Universal Robots PolyScope program: weigh_touch3.urp

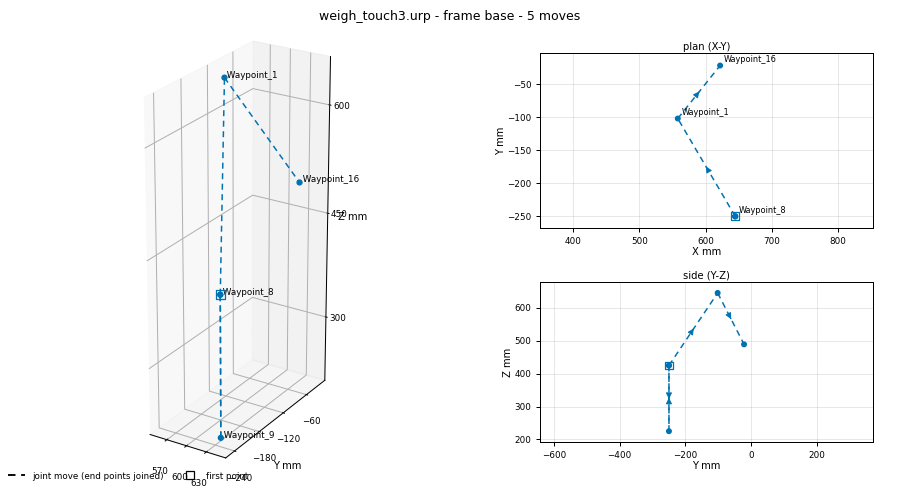
[picture p0: tool path of weigh_touch3.urp in frame base, 5 of 5 moves have a stored position in this frame; points joined in program order, loops and branches not executed]
Program weigh_touch3 (installation=default directory=/programs/Nicolas_Arteaga/quality createdIn=5.8.2.10297 lastSavedIn=5.12.4.1101661 robotSerialNumber=20225502378)
Calibrated DH parameters: a=[0.00022, -0.425328, -0.389701, 0.000059, 0.000065, 0]; d=[0.162608, 0.803456, 9.992211, -10.662202, 0.099702, 0.099559]; alpha=[1.570756, 0.001543, 0.004316, 1.570651, -1.570122, 0]; deltaTheta=[0, 0.002917, 0.116094, -0.119008, 0, -0.000001]
Robot Program (runOnlyOnce=true)
  MoveJ speed 60 deg/s, acceleration 80 deg/s^2 (useActiveTCP=true) feature=Base
    Waypoint Waypoint_8: TCP in base x=644.963 y=-250.234 z=424.745 mm, rx=-0.4223 ry=1.4905 rz=0.4378 rad; joints [121.021, -52.336, 61.566, 67.994, -2.525, 192.758] deg; TCP offset x=0 y=0 z=191.5 mm, rx=0 ry=0 rz=0 rad
    Waypoint Waypoint_9: TCP in base x=644.964 y=-250.243 z=224.998 mm, rx=-0.4223 ry=1.4905 rz=0.4378 rad; joints [121.04, -41.53, 74.294, 46.989, -2.465, 190.226] deg
    Waypoint Waypoint_8: TCP in base x=644.963 y=-250.234 z=424.745 mm, rx=-0.4223 ry=1.4905 rz=0.4378 rad; joints [121.021, -52.336, 61.566, 67.994, -2.525, 192.758] deg
    Waypoint Waypoint_1: TCP in base x=557.994 y=-102.204 z=645.214 mm, rx=-1.3174 ry=0.9174 rz=-0.5836 rad; joints [121.342, -85.625, 61.567, 24.73, -2.556, 192.757] deg
    Waypoint Waypoint_16: TCP in base x=622.09 y=-21.999 z=488.949 mm, rx=0.729 ry=1.5781 rz=1.7949 rad; joints [135.515, -94.567, 106.176, -67.801, 9.2, 55.784] deg
    'Move to final position'
